TYPE ST_PNInput_Battery :
STRUCT
	ui_SocMinLimit	:	UINT	:=	100;
	ui_SocMaxLimit	:	UINT	:=	0;
END_STRUCT
END_TYPE

(* stored: Version 1.1.0.1, ProductVersion 3.1.4024.12
   DUT ST_PNInput_Battery: Id {a4d61282-7f77-4188-9130-09f98a2cc63e} *)
